INTERFACE I_DeserializerArrayForwardEnumerator EXTENDS I_Disposable

PROPERTY PUBLIC Current : I_Deserializer
GET
END_GET
END_PROPERTY

PROPERTY Index : DINT
GET
END_GET
END_PROPERTY

PROPERTY IsValid : BOOL
GET
END_GET
END_PROPERTY

METHOD MoveNext : BOOL
VAR_INPUT
END_VAR
END_METHOD

END_INTERFACE

(* stored: Version 1.1.0.1, ProductVersion 3.1.4024.12
   Itf I_DeserializerArrayForwardEnumerator: Id {8cb67853-395c-0f99-1f7b-67029af57b91}
   Property Current: Id {3d35568c-0718-0c13-3e79-5f1471e5a412}
   Get Get: Id {198d9588-6c53-01c5-2e6e-e660545231be}
   Property Index: Id {be569162-232c-056d-0b97-291932ea06d2}
   Get Get: Id {7ad649fc-1331-0671-2f7f-8de762c8c982}
   Property IsValid: Id {2f7501cd-25e3-0f70-3fc7-fa43a085e4e6}
   Get Get: Id {7c5cc91d-5f33-06ca-1a27-857c6eaaa75c}
   Method MoveNext: Id {5c58b2c4-affc-0676-34e2-907709e3ebee} *)
